DATA_BLOCK "DB_ProfinetDiagnostic"
TITLE = DB_ProfinetDiagnostic
{ S7_Optimized_Access := 'TRUE' }
AUTHOR : MHSE
FAMILY : GeneralSystemFunctions
VERSION : 3.0
NON_RETAIN
//Data block to store profinet network diagnostic data.
   VAR
      ProfinetNetworks { ExternalAccessible := 'False'; ExternalVisible := 'False'; ExternalWritable := 'False'; S7_SetPoint := 'False'} : Array[1..10] of "UDT_ProfinetNetwork";
   END_VAR


BEGIN

END_DATA_BLOCK

DATA_BLOCK "DI_OnOffDevices"
{ S7_Optimized_Access := 'TRUE' }
AUTHOR : MHSE
FAMILY : GeneralSystemFunctions
VERSION : 2.0
NON_RETAIN
"FB_OnOffDevices"

BEGIN

END_DATA_BLOCK

DATA_BLOCK "DB_Statistics"
TITLE = DB_Statistics
{ S7_Optimized_Access := 'TRUE' }
AUTHOR : MHSE
FAMILY : GeneralSystemFunctions
VERSION : 3.0
NON_RETAIN
//Data block to store statistical data.
   VAR
      Communication : Struct   // Communication statistic
         TCPIPConnect : "UDT_TCPIPConnectStatistics";   // TCPIP Connect statistics
         TCPIPReceive : "UDT_TCPIPReceiveStatistics";   // TCPIP Receive statistics
      END_STRUCT;
      System : Struct   // System statistic
         MCP { S7_SetPoint := 'False'} : "UDT_MainControlPanelStatistics";   // Statistics of Main Control Panel
         CPG01 : "UDT_ControlPowerGroupStatistics";   // Statistics of  Control Power Group 01
         CPG02 : "UDT_ControlPowerGroupStatistics";   // Statistics of  Control Power Group 02
         CPG03 : "UDT_ControlPowerGroupStatistics";   // Statistics of  Control Power Group 03
         CPG04 : "UDT_ControlPowerGroupStatistics";   // Statistics of  Control Power Group 04
         CPG05 : "UDT_ControlPowerGroupStatistics";   // Statistics of  Control Power Group 05
         Profinet { S7_SetPoint := 'False'} : "UDT_ProfiDiagStatistics";
      END_STRUCT;
   END_VAR


BEGIN

END_DATA_BLOCK

DATA_BLOCK "DB_FIFOMedPrioMsg"
TITLE = DB_FIFO
{ S7_Optimized_Access := 'TRUE' }
AUTHOR : MHSE
FAMILY : GeneralSystemFunctions
VERSION : 3.0
NON_RETAIN
//Data block to store FIFO registers.
   VAR RETAIN
      Header { ExternalAccessible := 'False'; ExternalVisible := 'False'; ExternalWritable := 'False'; S7_SetPoint := 'False'} : "UDT_FifoHeader";   // FIFO Header
      Data { ExternalAccessible := 'False'; ExternalVisible := 'False'; ExternalWritable := 'False'; S7_SetPoint := 'False'} : Array[0..199] of "UDT_Message";   // FIFO data buffer
   END_VAR


BEGIN

END_DATA_BLOCK

DATA_BLOCK "DB_FIFOLowPrioMsg"
TITLE = DB_FIFO
{ S7_Optimized_Access := 'TRUE' }
AUTHOR : MHSE
FAMILY : GeneralSystemFunctions
VERSION : 3.0
NON_RETAIN
//Data block to store FIFO registers.
   VAR RETAIN
      Header { ExternalAccessible := 'False'; ExternalVisible := 'False'; ExternalWritable := 'False'; S7_SetPoint := 'False'} : "UDT_FifoHeader";   // FIFO Header
      Data { ExternalAccessible := 'False'; ExternalVisible := 'False'; ExternalWritable := 'False'; S7_SetPoint := 'False'} : Array[0..199] of "UDT_Message";   // FIFO data buffer
   END_VAR


BEGIN

END_DATA_BLOCK

DATA_BLOCK "DB_FIFORcvMsg"
TITLE = DB_FIFO
{ S7_Optimized_Access := 'TRUE' }
AUTHOR : MHSE
FAMILY : GeneralSystemFunctions
VERSION : 3.0
NON_RETAIN
//Data block to store FIFO registers.
   VAR RETAIN
      Header { ExternalAccessible := 'False'; ExternalVisible := 'False'; ExternalWritable := 'False'; S7_SetPoint := 'False'} : "UDT_FifoHeader";   // FIFO Header
      Data { ExternalAccessible := 'False'; ExternalVisible := 'False'; ExternalWritable := 'False'; S7_SetPoint := 'False'} : Array[0..199] of "UDT_Message";   // FIFO data buffer
   END_VAR


BEGIN

END_DATA_BLOCK

DATA_BLOCK "DB_ParametrizationErrors"
TITLE = DB_ParametrizationErrors
{ S7_Optimized_Access := 'TRUE' }
AUTHOR : MHSE
FAMILY : GeneralSystemFunctions
VERSION : 3.0
NON_RETAIN
//Data block to store parametrization errors.
   VAR
      System { ExternalAccessible := 'False'; ExternalVisible := 'False'; ExternalWritable := 'False'} : Struct
         Communication { ExternalAccessible := 'False'; ExternalVisible := 'False'; ExternalWritable := 'False'} : Struct
            TCPIPSendError { ExternalAccessible := 'False'; ExternalVisible := 'False'; ExternalWritable := 'False'} : Bool;   // TCPIP send error
            TCPIPSendWarning { ExternalAccessible := 'False'; ExternalVisible := 'False'; ExternalWritable := 'False'} : Bool;   // TCPIP send warning
            TCPIPReceiveError { ExternalAccessible := 'False'; ExternalVisible := 'False'; ExternalWritable := 'False'} : Bool;   // TCPIP receive error
            TCPIPReceiveWarning { ExternalAccessible := 'False'; ExternalVisible := 'False'; ExternalWritable := 'False'} : Bool;   // TCPIP receive warning
         END_STRUCT;
      END_STRUCT;
   END_VAR


BEGIN

END_DATA_BLOCK

DATA_BLOCK "DB_CommonStatus"
TITLE = DB_Status
{ S7_Optimized_Access := 'TRUE' }
AUTHOR : MHSE
FAMILY : GeneralSystemFunctions
VERSION : 3.0
NON_RETAIN
//Data block to store status data.
   VAR
      Communication : Struct   // Communication status
         TCPIPConnect : "UDT_CommonStatus";   // FB_TCPIPConnect status
      END_STRUCT;
      System : Struct   // System statuses
         System1 { S7_SetPoint := 'False'} : "UDT_CommonStatus";
         MCP { S7_SetPoint := 'False'} : "UDT_CommonStatus";
         CPG01 : "UDT_CommonStatus";
         CPG02 : "UDT_CommonStatus";
         CPG03 : "UDT_CommonStatus";
         CPG04 : "UDT_CommonStatus";
         CPG05 : "UDT_CommonStatus";
         test { S7_SetPoint := 'True'} : Int;
      END_STRUCT;
   END_VAR


BEGIN

END_DATA_BLOCK

DATA_BLOCK "DB_Status"
TITLE = DB_Status
{ S7_Optimized_Access := 'TRUE' }
AUTHOR : MHSE
FAMILY : GeneralSystemFunctions
VERSION : 3.0
NON_RETAIN
//Data block to store status data.
   VAR
      Communication : Struct   // Communication status
         TCPIPConnect : "UDT_TCPIPConnectStatus";   // FB_TCPIPConnect status
      END_STRUCT;
      System : Struct   // System status
         MCP { S7_SetPoint := 'False'} : "UDT_MainControlPanelStatus";   // Status of Main Control Panel
         CPG01 : "UDT_ControlPowerGroupStatus";   // Status of  Control Power Group 01
         CPG02 : "UDT_ControlPowerGroupStatus";   // Status of  Control Power Group 02
         CPG03 : "UDT_ControlPowerGroupStatus";   // Status of  Control Power Group 03
         CPG04 : "UDT_ControlPowerGroupStatus";   // Status of  Control Power Group 04
         CPG05 : "UDT_ControlPowerGroupStatus";   // Status of  Control Power Group 05
         System1 : "UDT_SystemControlStatus";
      END_STRUCT;
   END_VAR


BEGIN

END_DATA_BLOCK

FUNCTION_BLOCK "FB_SoftVersion"
TITLE = FB_SoftVersion
{ S7_Optimized_Access := 'TRUE' }
AUTHOR : MHSE
FAMILY : GeneralSystemFunctions
VERSION : 3.0
// ATTRIBUTES
// AUTO_NUMBER = True
// BLOCK_NUMBER = 28
// END_ATTRIBUTES
//Function block to get the program checksums.
   VAR_INPUT
      is_ActualDateTime : String;   // Actual date and time
   END_VAR

   VAR_OUTPUT
      qs_SoftVersion : String[8];   // Software version
      qa_StandardCRC : Array[0..7] of Byte;   // Standard program checksum output
      qa_SafetyCRC : Array[0..7] of Byte;   // Safety program checksum output
   END_VAR

   VAR
      sFB_GetChecksum_Safety {InstructionName := 'GetChecksum'; LibVersion := '1.0'} : GetChecksum;   // Safety checksum read block
      sFB_GetChecksum_Standard {InstructionName := 'GetChecksum'; LibVersion := '1.0'} : GetChecksum;   // Standard checksum read block
   END_VAR
   VAR RETAIN
      sa_StandardCRC : Array[0..7] of Byte;   // Standard program checksum
      sa_SafetyCRC : Array[0..7] of Byte;   // Safety program checksum
   END_VAR
   VAR
      sa_NewStandardCRC { ExternalAccessible := 'False'; ExternalVisible := 'False'; ExternalWritable := 'False'} : Array[0..7] of Byte;   // New standard program checksum
      sa_NewSafetyCRC { ExternalAccessible := 'False'; ExternalVisible := 'False'; ExternalWritable := 'False'} : Array[0..7] of Byte;   // New safety program checksum
   END_VAR
   VAR RETAIN
      ss_Date { ExternalAccessible := 'False'; ExternalVisible := 'False'; ExternalWritable := 'False'} : String[8];   // Date charater string
   END_VAR

   VAR_TEMP
      ta_StandardCRC : Struct   // GetChecksum
         tx_Done : Bool;   // GetChecksum - Done
         tx_Busy : Bool;   // GetChecksum - Busy
         tx_Error : Bool;   // GetChecksum - Error
         tw_Status : Word;   // GetChecksum - Status
      END_STRUCT;
      ta_SafetyCRC : Struct   // GetChecksum
         tx_Done : Bool;   // GetChecksum - Done
         tx_Busy : Bool;   // GetChecksum - Busy
         tx_Error : Bool;   // GetChecksum - Error
         tw_Status : Word;   // GetChecksum - Status
      END_STRUCT;
      tx_CRCValid : Bool;   // Checksums valid
   END_VAR


BEGIN
	(*
	----------------------------------------------------------------------------------------

	Version history:
	Date        | Version   | Author        | Remark
	----------------------------------------------------------------------------------------
	24/05/2019  | 0.1       | K.Pokorski    | first release MHS TIA 15.1
	14/06/2019  | 0.2       | A.Nowak       | Replacement of instruction if for direct write into variable - Region 2
	24/07/2019  | 2.0       | L.Klar        | 2.0 MHS library release TIA 15.1
	27/08/2019  | 2.2       | K.Pokorski    | Comments adjusted
	12/11/2019  | 3.0       | P.Majka       | 3.0 MHS library release TIA 15.1
	21/02/2023  | 4.0       | F.Baten       | 4.0 Release TIA 17.5
	*)

	REGION 1 - Standard and safety program checksums

	    // Scope - 1 - Standard program CRC
	    #sFB_GetChecksum_Standard(Scope := 1,
	                              Done => #ta_StandardCRC.tx_Done,
	                              Busy => #ta_StandardCRC.tx_Busy,
	                              Error => #ta_StandardCRC.tx_Error,
	                              Status => #ta_StandardCRC.tw_Status,
	                              Checksum := #sa_NewStandardCRC);

	    // Scope - 2 - Safety program CRC
	    #sFB_GetChecksum_Safety(Scope := 2,
	                            Done => #ta_SafetyCRC.tx_Done,
	                            Busy => #ta_SafetyCRC.tx_Busy,
	                            Error => #ta_SafetyCRC.tx_Error,
	                            Status => #ta_SafetyCRC.tw_Status,
	                            Checksum := #sa_NewSafetyCRC);

	END_REGION

	REGION 2 - Checksums comparison

	    #tx_CRCValid := (#sa_NewStandardCRC = #sa_StandardCRC)
	    AND (#sa_SafetyCRC = #sa_NewSafetyCRC);

	END_REGION

	REGION 3 - New software version

	    // Separate the year, mounth and day from actual date and time and connect it to one string
	    IF (NOT #tx_CRCValid)                                           // Checksums not valid
	    THEN

	        #ss_Date := CONCAT(IN1 := MID(IN := #is_ActualDateTime,
	                                                         L := 4,
	                                                         P := 1),

	                           IN2 := MID(IN := #is_ActualDateTime,
	                                      L := 2,
	                                      P := 6),

	                           IN3 := MID(IN := #is_ActualDateTime,
	                                      L := 2,
	                                      P := 9));

	        // Standard progrm checksum update
	        #sa_StandardCRC := #sa_NewStandardCRC;

	        // Safety program checksum update
	        #sa_SafetyCRC := #sa_NewSafetyCRC;

	    END_IF;

	END_REGION

	REGION 4 - Write outputs

	    // New program date
	    #qs_SoftVersion := #ss_Date;

	    // Actual standard program checksum
	    #qa_StandardCRC := #sa_StandardCRC;

	    // Actual safety program checksum
	    #qa_SafetyCRC := #sa_SafetyCRC;

	END_REGION
END_FUNCTION_BLOCK

DATA_BLOCK "DB_Configuration"
TITLE = DB_Configuration
{ S7_Optimized_Access := 'TRUE' }
AUTHOR : MHSE
FAMILY : GeneralSystemFunctions
VERSION : 3.0
NON_RETAIN
//Data block to store configuration data.
   VAR RETAIN
      System { ExternalAccessible := 'False'; ExternalVisible := 'False'; ExternalWritable := 'False'} : Struct   // System configuration
         Connection { ExternalAccessible := 'False'; ExternalVisible := 'False'; ExternalWritable := 'False'} : "UDT_Connection";   // Connection configuration
      END_STRUCT;
   END_VAR


BEGIN
   System.Connection.ActiveEstablished := TRUE;
   System.Connection.Interface_ID := 64;
   System.Connection.ID := 16#0001;
   System.Connection.IP[1] := 192;
   System.Connection.IP[2] := 168;
   System.Connection.IP[3] := 3;
   System.Connection.IP[4] := 53;
   System.Connection.Port := 42300;
   System.Connection.ConTimeout := 5000;

END_DATA_BLOCK

FUNCTION_BLOCK "FB_ProfiDiag"
TITLE = FB_ProfiDiag
{ S7_Optimized_Access := 'TRUE' }
AUTHOR : MHSE
FAMILY : GeneralSystemFunctions
VERSION : 3.0
// ATTRIBUTES
// AUTO_NUMBER = True
// BLOCK_NUMBER = 25
// END_ATTRIBUTES
//Function block to diagnose Profinet network.
   VAR_INPUT
      iui_LADDR : HW_IOSYSTEM;   // Hardware identifier of the PROFINET IO
      ix_ExternalScan { ExternalAccessible := 'False'; ExternalVisible := 'False'; ExternalWritable := 'False'} : Bool;   // External scan
   END_VAR

   VAR_OUTPUT
      qx_ProfinetOk { ExternalAccessible := 'False'; ExternalVisible := 'False'; ExternalWritable := 'False'} : Bool;   // Profinet ok
      qx_Error { ExternalAccessible := 'False'; ExternalVisible := 'False'; ExternalWritable := 'False'} : Bool;   // Collective error output
   END_VAR

   VAR_IN_OUT
      iqUDT_EquipmentControl : "UDT_EquipmentControl";   // Equipment control structure
      iqUDT_PNDiagArray : "UDT_ProfinetNetwork";   // Profinet devices status array
      iqUDT_Statistics : "UDT_ProfiDiagStatistics";   // Statistics structure
   END_VAR

   VAR
      s_GetProjectName {InstructionName := 'Get_Name'; LibVersion := '1.3'} : Get_Name;   // Get name function
      sa_Status : Struct   // Status structure
         ErrorCode : Struct   // Error code structure
            DeviceState : Int;   // Siemens "DeviceState" error code
            GEO2LOG : Int;   // Siemens "GEO2LOG" error code
            LOG2GEO : Int;   // Siemens "LOG2GEO" error code
            GetName : Word;   // Siemens "GetName" error code
         END_STRUCT;
      END_STRUCT;
      sx_PNOK : Bool := FALSE;   // Profinet OK
      sx_NewEvent { ExternalAccessible := 'False'; ExternalVisible := 'False'; ExternalWritable := 'False'} : Bool;   // New event
   END_VAR

   VAR_TEMP
      tv_ProfinetGeoAdr {InstructionName := 'GEOADDR'; LibVersion := '1.0'} : GEOADDR;   // Profinet network geo structure
      tv_DeviceGeoAdr {InstructionName := 'GEOADDR'; LibVersion := '1.0'} : GEOADDR;   // Profinet device geo structure
      ta_Configured : Array[0..1024] of Bool;   // Configured devices array
      ta_Exist : Array[0..1024] of Bool;   // Existing devices array
      ta_Error : Array[0..1024] of Bool;   // Devices errors array
      ti_DeviceNr : Int;   // Device number
      ti_NrOfDevicesError : Int;   // Number of devices error
      ti_DiagArraySize : Int;   // Diagnostic array size
   END_VAR

   VAR CONSTANT
      cui_ConfiguredDevicesMode : UInt := 1;   // Scan mode of configured devices
      cui_ExistingDevicesMode : UInt := 4;   // Scan mode of existing devices
      cui_DevicesErrorMode : UInt := 2;   // Scan mode of devices error
      cui_HWType : UInt := 2;   // IO device hardware type
      cui_Area : UInt := 1;   // IO device area
   END_VAR


BEGIN
	(*
	----------------------------------------------------------------------------------------

	Version history:
	Date        | Version   | Author        | Remark
	----------------------------------------------------------------------------------------
	24/05/2019  | 0.1       | K.Pokorski    | first release MHS TIA 15.1
	13/06/2019  | 0.2       | A.Nowak       | Replacement of instruction if for direct write into variable - Region 3
	24/06/2019  | 0.3       | L.Klar        | Status running added
	19/07/2019  | 0.5       | L.Klar        | Status handling changed, output qx_ProfinetOk added
	24/07/2019  | 2.0       | L.Klar        | 2.0 MHS library release TIA 15.1
	14/08/2019  | 2.1       | K.Pokorski    | HW_ID and TIA device project name handling added
	26/08/2019  | 2.2       | K.Pokorski    | Comments adjusted
	20/09/2019  | 2.3       | K.Pokorski    | "UDT_Status" deleted
	04/11/2019  | 2.4       | L.Klar        | Scan profinet and first scan changed from memory bit to DB variable
	12/11/2019  | 3.0       | P.Majka       | 3.0 MHS library release TIA 15.1
	21/02/2023  | 4.0       | F.Baten       | 4.0 Release TIA 17.5
	*)

	REGION 1 – Scan request

	    IF ("DB_Memory".ScanProfinet    // Scan request from diagnostic OB
	        OR "DB_Memory".FirstScan    // First PLC cycle
	        OR #ix_ExternalScan)        // External scan available
	    THEN

	        #sx_PNOK := FALSE;

	    END_IF;

	END_REGION

	REGION 2 – Devices states update

	    // Scan devices, extract device status: configured, exists, error when profinet network not ok
	    IF (NOT #sx_PNOK)       // Profinet needs a scan
	    THEN

	        #sa_Status.ErrorCode.DeviceState := DeviceStates(LADDR := #iui_LADDR,
	                                                         MODE := #cui_ConfiguredDevicesMode,
	                                                         STATE := #ta_Configured);

	        #sa_Status.ErrorCode.DeviceState := DeviceStates(LADDR := #iui_LADDR,
	                                                         MODE := #cui_ExistingDevicesMode,
	                                                         STATE := #ta_Exist);

	        #sa_Status.ErrorCode.DeviceState := DeviceStates(LADDR := #iui_LADDR,
	                                                         MODE := #cui_DevicesErrorMode,
	                                                         STATE := #ta_Error);

	    END_IF;

	END_REGION

	REGION 3 – Devices Statuses update

	    // Move device state to diagnostic structure if network required scan and no error occured during scan
	    IF (NOT #sx_PNOK                                                                                                    // Profinet not ok
	        AND #sa_Status.ErrorCode.DeviceState = 0)                                                                       // "DeviceStates" error free
	    THEN

	        // Initialise reset device errors counter
	        #ti_NrOfDevicesError := 0;

	        // Maximum number of Profinet devices
	        #ti_DiagArraySize := "FC_GetNrOfArrayEl"(iv_Array := #iqUDT_PNDiagArray.DeviceStatus);

	        // A loop operating on Profinet devices
	        FOR #ti_DeviceNr := 0 TO (#ti_DiagArraySize - 1)
	        DO

	            // The device is configured in TIA Portal
	            IF (#ta_Configured[#ti_DeviceNr])                                                                           // Devices configured
	            THEN

	                // Set the device configured status bit in diagnostic structure
	                #iqUDT_PNDiagArray.DeviceStatus[#ti_DeviceNr].DeviceState.Configure := TRUE;

	                // Move device profinet number to diagnostic structure
	                #iqUDT_PNDiagArray.DeviceStatus[#ti_DeviceNr].DeviceState.ProfinetNumber := INT_TO_UINT(#ti_DeviceNr);

	                // Get the Profinet network IOSystem address
	                #sa_Status.ErrorCode.LOG2GEO := LOG2GEO(LADDR := #iui_LADDR, GEOADDR := #tv_ProfinetGeoAdr);

	                // Configuring parameters for extracting the device's HW_ID
	                #tv_DeviceGeoAdr.HWTYPE := #cui_HWType;
	                #tv_DeviceGeoAdr.AREA := #cui_Area;
	                #tv_DeviceGeoAdr.STATION := INT_TO_UINT(#ti_DeviceNr);
	                #tv_DeviceGeoAdr.IOSYSTEM := #tv_ProfinetGeoAdr.IOSYSTEM;

	                // Extracting the device's HW_ID
	                #sa_Status.ErrorCode.GEO2LOG := GEO2LOG(GEOADDR := #tv_DeviceGeoAdr,
	                                                        LADDR => #iqUDT_PNDiagArray.DeviceStatus[#ti_DeviceNr].DeviceState.HW_ID);

	                // Move device's project name to diagnostic structure
	                #s_GetProjectName(LADDR := #iui_LADDR,
	                                  STATION_NR := INT_TO_UINT(#ti_DeviceNr),
	                                  STATUS => #sa_Status.ErrorCode.GetName,
	                                  DATA := #iqUDT_PNDiagArray.DeviceStatus[#ti_DeviceNr].DeviceState.PNDeviceName);

	                // Move device exist state to the Profinet diagnostic structure
	                IF (#ta_Exist[#ti_DeviceNr])                                                                                // Device exist
	                THEN

	                    #iqUDT_PNDiagArray.DeviceStatus[#ti_DeviceNr].DeviceState.Exist := TRUE;

	                ELSE

	                    #iqUDT_PNDiagArray.DeviceStatus[#ti_DeviceNr].DeviceState.Exist := FALSE;

	                    // Increment the number of devices error
	                    #ti_NrOfDevicesError += 1;

	                END_IF;
	                // Move device error state to the Profinet diagnostic structure
	                IF (NOT #ta_Error[#ti_DeviceNr])                                                                            // Device is error free
	                THEN

	                    #iqUDT_PNDiagArray.DeviceStatus[#ti_DeviceNr].DeviceState.Error := FALSE;

	                ELSE

	                    // New error detected
	                    #sx_NewEvent := NOT #iqUDT_PNDiagArray.DeviceStatus[#ti_DeviceNr].DeviceState.Error;

	                    // Statistics handling
	                    IF (#ta_Error[#ti_DeviceNr]                                                                             // Device has error
	                        OR #iqUDT_EquipmentControl.Command.ResetData)                                                      // Reset statistics available
	                    THEN

	                        "FC_Statistics"(ix_Reset := #iqUDT_EquipmentControl.Command.ResetData,
	                                        ix_Activate := #ta_Error[#ti_DeviceNr],
	                                        ix_RTrigActivate := #sx_NewEvent,
	                                        iqUDT_Statistics := #iqUDT_Statistics.DeviceError[#ti_DeviceNr]);

	                    END_IF;

	                    #iqUDT_PNDiagArray.DeviceStatus[#ti_DeviceNr].DeviceState.Error := TRUE;

	                    // Increment number of devices error
	                    #ti_NrOfDevicesError += 1;

	                END_IF;

	                // Reset all diagnostic information if the device is not configured in TIA Portal
	            ELSE

	                #iqUDT_PNDiagArray.DeviceStatus[#ti_DeviceNr].DeviceState.Configure := FALSE;
	                #iqUDT_PNDiagArray.DeviceStatus[#ti_DeviceNr].DeviceState.Exist := FALSE;
	                #iqUDT_PNDiagArray.DeviceStatus[#ti_DeviceNr].DeviceState.Error := FALSE;
	                #iqUDT_PNDiagArray.DeviceStatus[#ti_DeviceNr].DeviceState.HW_ID := 0;
	                #iqUDT_PNDiagArray.DeviceStatus[#ti_DeviceNr].DeviceState.ProfinetNumber := 0;
	                #iqUDT_PNDiagArray.DeviceStatus[#ti_DeviceNr].DeviceState.PNDeviceName := '';

	            END_IF;

	        END_FOR;

	    END_IF;

	END_REGION

	REGION 4 – Profinet OK

	    // Reset profinet error
	    IF (#ti_NrOfDevicesError = 0                        // Number of devices error equal to zero
	        AND (#iqUDT_EquipmentControl.Command.Reset     // Error reset required
	        OR #ix_ExternalScan))                           // External scan active
	    THEN

	        #sx_PNOK := TRUE;

	    END_IF;

	END_REGION

	REGION 5 – Status

	    // Update Profinet ok output status
	    #qx_ProfinetOk := #sx_PNOK;

	    // Create the collective block error bit
	    #qx_Error := #sa_Status.ErrorCode.DeviceState <> 0       // Profinet network error
	    OR #sa_Status.ErrorCode.GEO2LOG <> 0                     // "Geo2Log" standard Siemens block error
	    OR #sa_Status.ErrorCode.LOG2GEO <> 0                     // "Log2Geo" standard Siemens block error
	    OR #sa_Status.ErrorCode.GetName > 16#8000;               // "GetName" standard Siemens block error

	END_REGION
END_FUNCTION_BLOCK

FUNCTION "FC_Simulation" : Void
TITLE = FC_Simulation
{ S7_Optimized_Access := 'TRUE' }
AUTHOR : MHSE
FAMILY : GeneralSystemFunctions
VERSION : 3.0
// ATTRIBUTES
// AUTO_NUMBER = True
// BLOCK_NUMBER = 13
// END_ATTRIBUTES
//Function to enable simulation mode.
   VAR_TEMP
      tx_Done : Bool;
      tx_Error : Bool;
   END_VAR


BEGIN
	(*
	----------------------------------------------------------------------------------------

	Version history:
	Date        | Version   | Author        | Remark
	----------------------------------------------------------------------------------------
	24/05/2019  | 0.1       | L.Klar        | first release MHS TIA 15.1
	24/07/2019  | 2.0       | L.Klar        | 2.0 MHS library release TIA 15.1
	04/11/2019  | 2.1       | L.Klar        | Simulation bit changed from memory to DB variable
	12/11/2019  | 3.0       | P.Majka       | 3.0 MHS library release TIA 15.1
	21/02/2023  | 4.0       | F.Baten       | 4.0 Release TIA 17.5
	*)

	REGION 1 - Disabling and Enabling devices

	    "DI_OnOffDevices"(ix_Simulation := "DB_Memory".Simulation,
	                      qx_Done => #tx_Done,
	                      qx_Error => #tx_Error,
	                      iqa_ProfinetNetworks := "DB_ProfinetDiagnostic".ProfinetNetworks);

	END_REGION



END_FUNCTION

FUNCTION "FC_TimeToString" : Void
TITLE = FC_TimeToString
{ S7_Optimized_Access := 'TRUE' }
AUTHOR : MHSE
FAMILY : GeneralSystemFunctions
VERSION : 3.0
// ATTRIBUTES
// AUTO_NUMBER = True
// BLOCK_NUMBER = 29
// END_ATTRIBUTES
//Function to convert date in DTL to the string format.
   VAR_INPUT
      ia_Date {InstructionName := 'DTL'; LibVersion := '1.0'} : DTL;   // DTL format date
   END_VAR

   VAR_OUTPUT
      qs_Date : String;   // String format date
   END_VAR

   VAR_TEMP
      ta_StringDate : Struct   // String format date
         Year : String;   //   Year
         Month : String[2];   //   Month
         Day : String[2];   //   Day
         Hour : String[2];   //   Hour
         Minute : String[2];   //   Minunte
         Second : String[2];   //   Second
         Millisecond : String[4];   //   Millisecond
      END_STRUCT;
      ta_HTAReturn : Struct   // HTA operation status
         Year : Word;   //   Year
         Month : Word;   //   Month
         Day : Word;   //   Day
         Hour : Word;   //   Hour
         Minute : Word;   //   Minunte
         Second : Word;   //   Second
         Millisecond : Word;   //   Millisecond
      END_STRUCT;
   END_VAR

   VAR CONSTANT
      ci_Positions4 : USInt := 4;   // Number of character positions
      ci_DecimalPlaces0 : USInt := 0;   // Number of decimal places
      ci_Format0 : USInt := 0;   // Output format of the characters
      ci_Position1 : USInt := 1;   // Character starting at which the result is written
      cc_Colon : Char := ':';   // Colon sign
   END_VAR


BEGIN
	(*
	----------------------------------------------------------------------------------------

	Version history:
	Date        | Version   | Author        | Remark
	----------------------------------------------------------------------------------------
	24/05/2019  | 0.1       | K.Pokorski    | first release MHS TIA 15.1
	24/07/2019  | 2.0       | L.Klar        | 2.0 MHS library release TIA 15.1
	27/08/2019  | 2.1       | M.Kurpiers    | Comments adjusted
	05/09/2019  | 2.2       | K.Pokorski    | FC changed from unoptimized to optimized
	12/11/2019  | 3.0       | P.Majka       | 3.0 MHS library release TIA 15.1
	16/02/2023  | 3.1       | F.Baten       | Added constants
	21/02/2023  | 4.0       | F.Baten       | 4.0 Release TIA 17.5
	*)

	REGION 1 - Date and time separation

	    // Convert the year into a character string
	    VAL_STRG(IN := #ia_Date.YEAR,
	             SIZE := #ci_Positions4,
	             PREC := #ci_DecimalPlaces0,
	             FORMAT := USINT_TO_WORD(#ci_Format0),
	             P := #ci_Position1,
	             OUT => #ta_StringDate.Year);

	    // Using the HTA function, convert date into a string format
	    #ta_HTAReturn.Month := HTA(IN := WORD_TO_BYTE(INT_TO_BCD16((USINT_TO_INT(#ia_Date.MONTH)))), N := 1, OUT => #ta_StringDate.Month);                          // Convert the month
	    #ta_HTAReturn.Day := HTA(IN := WORD_TO_BYTE(INT_TO_BCD16((USINT_TO_INT(#ia_Date.DAY)))), N := 1, OUT => #ta_StringDate.Day);                                // Convert the day
	    #ta_HTAReturn.Hour := HTA(IN := WORD_TO_BYTE(INT_TO_BCD16((USINT_TO_INT(#ia_Date.HOUR)))), N := 1, OUT => #ta_StringDate.Hour);                             // Convert the hour
	    #ta_HTAReturn.Minute := HTA(IN := WORD_TO_BYTE(INT_TO_BCD16((USINT_TO_INT(#ia_Date.MINUTE)))), N := 1, OUT => #ta_StringDate.Minute);                       // Convert the minute
	    #ta_HTAReturn.Second := HTA(IN := WORD_TO_BYTE(INT_TO_BCD16((USINT_TO_INT(#ia_Date.SECOND)))), N := 1, OUT => #ta_StringDate.Second);                       // Convert the second
	    #ta_HTAReturn.Millisecond := HTA(IN := INT_TO_BCD16((UDINT_TO_INT(#ia_Date.NANOSECOND / 1000000))), N := 2, OUT => #ta_StringDate.Millisecond);              // Convert the millisecond

	END_REGION

	REGION 2 - Timestamp preparation

	    // Combine several input strings into one long output string
	    #qs_Date := (CONCAT(IN1 := #ta_StringDate.Year,
	                        IN2 := #cc_Colon,
	                        IN3 := #ta_StringDate.Month,
	                        IN4 := #cc_Colon,
	                        IN5 := #ta_StringDate.Day,
	                        IN6 := #cc_Colon,
	                        IN7 := #ta_StringDate.Hour,
	                        IN8 := #cc_Colon,
	                        IN9 := #ta_StringDate.Minute,
	                        IN10 := #cc_Colon,
	                        IN11 := #ta_StringDate.Second,
	                        IN12 := #cc_Colon,
	                        IN13 := RIGHT(IN := #ta_StringDate.Millisecond, L := 3)));

	END_REGION
END_FUNCTION

DATA_BLOCK "DI_TCPIPReceive"
{ S7_Optimized_Access := 'TRUE' }
VERSION : 0.1
NON_RETAIN
"FB_TCPIPReceive"

BEGIN

END_DATA_BLOCK

DATA_BLOCK "DB_Time"
TITLE = DB_Time
{ S7_Optimized_Access := 'TRUE' }
AUTHOR : MHSE
FAMILY : GeneralSystemFunctions
VERSION : 3.0
NON_RETAIN
//Data block to store date and time data.
   VAR
      ActualTimeDTL {InstructionName := 'DTL'; LibVersion := '1.0'; ExternalAccessible := 'False'; ExternalVisible := 'False'; ExternalWritable := 'False'} : DTL;   // Actual date and time in DTL
      ActualTime { ExternalAccessible := 'False'; ExternalVisible := 'False'; ExternalWritable := 'False'} : String;   // Actual date and time in String
      Timestamp { ExternalAccessible := 'False'; ExternalVisible := 'False'; ExternalWritable := 'False'} : String[17];   // Actual date and time in String
      DaylightSaving { ExternalAccessible := 'False'; ExternalVisible := 'False'; ExternalWritable := 'False'} : Int;
   END_VAR


BEGIN

END_DATA_BLOCK

DATA_BLOCK "DI_TCPIPSend"
{ S7_Optimized_Access := 'TRUE' }
VERSION : 0.1
NON_RETAIN
"FB_TCPIPSend"

BEGIN

END_DATA_BLOCK

DATA_BLOCK "DB_SoftwareVersion"
TITLE = DB_SoftwareVersion
{ S7_Optimized_Access := 'TRUE' }
AUTHOR : MHSE
FAMILY : GeneralSystemFunctions
VERSION : 3.0
NON_RETAIN
//Data block to store software version data.
   VAR
      "Version" { ExternalAccessible := 'False'; ExternalVisible := 'False'; ExternalWritable := 'False'} : String[8];   // Software version
      StandardChecksum { ExternalAccessible := 'False'; ExternalVisible := 'False'; ExternalWritable := 'False'} : Array[0..7] of Byte;   // Standard program checksum
      SafetyChecksum { ExternalAccessible := 'False'; ExternalVisible := 'False'; ExternalWritable := 'False'} : Array[0..7] of Byte;   // Safety program checksum
   END_VAR


BEGIN

END_DATA_BLOCK

DATA_BLOCK "DB_Control"
{ S7_Optimized_Access := 'TRUE' }
AUTHOR : MHSE
FAMILY : Equimpent
VERSION : 0.1
NON_RETAIN
   VAR
      System1 { ExternalAccessible := 'False'; ExternalVisible := 'False'; ExternalWritable := 'False'; S7_SetPoint := 'False'} : "UDT_EquipmentControl";
   END_VAR


BEGIN

END_DATA_BLOCK

DATA_BLOCK "DB_FIFOHighPrioMsg"
TITLE = DB_FIFO
{ S7_Optimized_Access := 'TRUE' }
AUTHOR : MHSE
FAMILY : GeneralSystemFunctions
VERSION : 3.0
NON_RETAIN
//Data block to store FIFO registers.
   VAR
      Header { ExternalAccessible := 'False'; ExternalVisible := 'False'; ExternalWritable := 'False'; S7_SetPoint := 'False'} : "UDT_FifoHeader";   // FIFO Header
      Data { ExternalAccessible := 'False'; ExternalVisible := 'False'; ExternalWritable := 'False'; S7_SetPoint := 'False'} : Array[0..199] of "UDT_Message";   // FIFO data buffer
   END_VAR


BEGIN

END_DATA_BLOCK

DATA_BLOCK "DI_TCPIPConnect"
{ S7_Optimized_Access := 'TRUE' }
VERSION : 0.1
NON_RETAIN
"FB_TCPIPConnect"

BEGIN

END_DATA_BLOCK

FUNCTION_BLOCK "FB_SystemFunctions"
TITLE = FB_SystemFunctions
{ S7_Optimized_Access := 'TRUE' }
AUTHOR : MHSE
FAMILY : GeneralSystemFunctions
VERSION : 3.0
// ATTRIBUTES
// AUTO_NUMBER = True
// BLOCK_NUMBER = 200
// END_ATTRIBUTES
//Function to execute system functions.
   VAR
      sFB_SoftVersion { ExternalAccessible := 'False'; ExternalVisible := 'False'; ExternalWritable := 'False'; S7_SetPoint := 'False'} : "FB_SoftVersion";   // Software version block instance
      sFB_ProfiDiag_Net1 { ExternalAccessible := 'False'; ExternalVisible := 'False'; ExternalWritable := 'False'; S7_SetPoint := 'False'} : "FB_ProfiDiag";   // Profinet diagnostic block instance
      sFB_ProfiDiag_Net2 { ExternalAccessible := 'False'; ExternalVisible := 'False'; ExternalWritable := 'False'; S7_SetPoint := 'False'} : "FB_ProfiDiag";   // Profinet diagnostic block instance
      sFB_ProfiDiag_Net3 { ExternalAccessible := 'False'; ExternalVisible := 'False'; ExternalWritable := 'False'; S7_SetPoint := 'False'} : "FB_ProfiDiag";   // Profinet diagnostic block instance
      sFB_ProfiDiag_Net4 { ExternalAccessible := 'False'; ExternalVisible := 'False'; ExternalWritable := 'False'; S7_SetPoint := 'False'} : "FB_ProfiDiag";   // Profinet diagnostic block instance
      sFB_ProfiDiag_Net5 { ExternalAccessible := 'False'; ExternalVisible := 'False'; ExternalWritable := 'False'; S7_SetPoint := 'False'} : "FB_ProfiDiag";   // Profinet diagnostic block instance
      sFB_ProfiDiag_Net6 { ExternalAccessible := 'False'; ExternalVisible := 'False'; ExternalWritable := 'False'; S7_SetPoint := 'False'} : "FB_ProfiDiag";   // Profinet diagnostic block instance
      sFB_ProfiDiag_Net7 { ExternalAccessible := 'False'; ExternalVisible := 'False'; ExternalWritable := 'False'; S7_SetPoint := 'False'} : "FB_ProfiDiag";   // Profinet diagnostic block instance
      sFB_ProfiDiag_Net8 { ExternalAccessible := 'False'; ExternalVisible := 'False'; ExternalWritable := 'False'; S7_SetPoint := 'False'} : "FB_ProfiDiag";   // Profinet diagnostic block instance
      sFB_ProfiDiag_Net9 { ExternalAccessible := 'False'; ExternalVisible := 'False'; ExternalWritable := 'False'; S7_SetPoint := 'False'} : "FB_ProfiDiag";   // Profinet diagnostic block instance
      sFB_ProfiDiag_Net10 { ExternalAccessible := 'False'; ExternalVisible := 'False'; ExternalWritable := 'False'; S7_SetPoint := 'False'} : "FB_ProfiDiag";   // Profinet diagnostic block instance
      sR_TRIG0_1Sec {InstructionName := 'R_TRIG'; LibVersion := '1.0'; ExternalAccessible := 'False'; ExternalVisible := 'False'; ExternalWritable := 'False'; S7_SetPoint := 'False'} : R_TRIG;   // Rise trigger to detect edge each 0.1 second
      sR_TRIG0_2Sec {InstructionName := 'R_TRIG'; LibVersion := '1.0'; ExternalAccessible := 'False'; ExternalVisible := 'False'; ExternalWritable := 'False'; S7_SetPoint := 'False'} : R_TRIG;   // Rise trigger to detect edge each 0.2 second
      sR_TRIG0_4Sec {InstructionName := 'R_TRIG'; LibVersion := '1.0'; ExternalAccessible := 'False'; ExternalVisible := 'False'; ExternalWritable := 'False'; S7_SetPoint := 'False'} : R_TRIG;   // Rise trigger to detect edge each 0.4 second
      sR_TRIG0_5Sec {InstructionName := 'R_TRIG'; LibVersion := '1.0'; ExternalAccessible := 'False'; ExternalVisible := 'False'; ExternalWritable := 'False'; S7_SetPoint := 'False'} : R_TRIG;   // Rise trigger to detect edge each 0.5 second
      sR_TRIG0_8Sec {InstructionName := 'R_TRIG'; LibVersion := '1.0'; ExternalAccessible := 'False'; ExternalVisible := 'False'; ExternalWritable := 'False'; S7_SetPoint := 'False'} : R_TRIG;   // Rise trigger to detect edge each 0.8 second
      sR_TRIG_1Sec {InstructionName := 'R_TRIG'; LibVersion := '1.0'; ExternalAccessible := 'False'; ExternalVisible := 'False'; ExternalWritable := 'False'; S7_SetPoint := 'False'} : R_TRIG;   // Rise trigger to detect edge each 1 second
      sR_TRIG1_6Sec {InstructionName := 'R_TRIG'; LibVersion := '1.0'; ExternalAccessible := 'False'; ExternalVisible := 'False'; ExternalWritable := 'False'; S7_SetPoint := 'False'} : R_TRIG;   // Rise trigger to detect edge each 1.6 second
      sR_TRIG_2Sec {InstructionName := 'R_TRIG'; LibVersion := '1.0'; ExternalAccessible := 'False'; ExternalVisible := 'False'; ExternalWritable := 'False'; S7_SetPoint := 'False'} : R_TRIG;   // Rise trigger to detect edge each 2 second
   END_VAR
   VAR DB_SPECIFIC
      sx_Reset { ExternalAccessible := 'False'; ExternalVisible := 'False'; ExternalWritable := 'False'} : Bool;   // Profinet fault reset
      sx_ResetData { ExternalAccessible := 'False'; ExternalVisible := 'False'; ExternalWritable := 'False'} : Bool;   // Profinet statistic data reset
   END_VAR
   VAR
      sx_Error { ExternalAccessible := 'False'; ExternalVisible := 'False'; ExternalWritable := 'False'} : Bool;
      sx_ProfiDiag_Net1_OK { ExternalAccessible := 'False'; ExternalVisible := 'False'; ExternalWritable := 'False'} : Bool;   // Profinet network 1 Ok
      sx_ProfiDiag_Net2_OK { ExternalAccessible := 'False'; ExternalVisible := 'False'; ExternalWritable := 'False'} : Bool;   // Profinet network 2 Ok
      sx_ProfiDiag_Net3_OK { ExternalAccessible := 'False'; ExternalVisible := 'False'; ExternalWritable := 'False'} : Bool;   // Profinet network 3 Ok
      sx_ProfiDiag_Net4_OK { ExternalAccessible := 'False'; ExternalVisible := 'False'; ExternalWritable := 'False'} : Bool;   // Profinet network 4 Ok
      sx_ProfiDiag_Net5_OK { ExternalAccessible := 'False'; ExternalVisible := 'False'; ExternalWritable := 'False'} : Bool;   // Profinet network 5 Ok
      sx_ProfiDiag_Net6_OK { ExternalAccessible := 'False'; ExternalVisible := 'False'; ExternalWritable := 'False'} : Bool;   // Profinet network 6 Ok
      sx_ProfiDiag_Net7_OK { ExternalAccessible := 'False'; ExternalVisible := 'False'; ExternalWritable := 'False'} : Bool;   // Profinet network 7 Ok
      sx_ProfiDiag_Net8_OK { ExternalAccessible := 'False'; ExternalVisible := 'False'; ExternalWritable := 'False'} : Bool;   // Profinet network 8 Ok
      sx_ProfiDiag_Net9_OK { ExternalAccessible := 'False'; ExternalVisible := 'False'; ExternalWritable := 'False'} : Bool;   // Profinet network 9 Ok
      sx_ProfiDiag_Net10_OK { ExternalAccessible := 'False'; ExternalVisible := 'False'; ExternalWritable := 'False'} : Bool;   // Profinet network 10 Ok
   END_VAR

   VAR_TEMP
      tui_LADDR : HW_IOSYSTEM;
      tUDT_EquipmentControl : "UDT_EquipmentControl";
      ti_RD_LOC_T_Status : Int;   // RD_LOC_T - Read actual date and time function status
      tx_replace : Bool;
   END_VAR


BEGIN
	(*
	----------------------------------------------------------------------------------------
	|                                                                                      |
	|  Copyright  2019             MHS                                                     |
	|  All Rights Reserved         Larenweg 90                                             |
	|                              5234 KC 's-Hertogenbosch,                               |
	|                              Netherlands                                             |
	|                                                                                      |
	----------------------------------------------------------------------------------------

	Version history:
	Date        | Version   | Author        | Remark
	----------------------------------------------------------------------------------------
	24/05/2019  | 0.1       | L.Klar        | first release MHS TIA 15.1
	24/07/2019  | 2.0       | L.Klar        | 2.0 MHS library release TIA 15.1
	03/10/2019  | 2.1       | L.Klar        | Comments adjusted
	04/10/2019  | 2.2       | L.Klar        | profinet scan marker reset added
	30/10/2019  | 2.3       | S.Theocharis  | Update the PN calls
	04/11/2019  | 2.4       | L.Klar        | Memory bits changed to DB variables
	12/11/2019  | 3.0       | P.Majka       | 3.0 MHS library release TIA 15.1
	11/12/2019  | 3.1       | S. Deulkar    | Called FC simulation in region 2
	21/02/2023  | 4.0       | F.Baten       | 4.0 Release TIA 17.5
	*)

	REGION 1 – PLC scan cycle measurement

	    "DB_Memory".PrevCycleTime := RUNTIME("DB_Memory".RuntimeMem) * 1000;

	END_REGION

	REGION 2 – Simulation

	    "FC_Simulation"();

	END_REGION

	REGION 3 – One shot of PLC clock pulse

	    // One shot every 0.1 sec of 10 Hz clock memory
	    #sR_TRIG0_1Sec(CLK := "DB_Memory".Clock_10Hz,
	                   Q => "DB_Memory"."OS_0.1sec");

	    // One shot every 0.2 sec of 5 Hz clock memory
	    #sR_TRIG0_2Sec(CLK := "DB_Memory".Clock_5Hz,
	                   Q => "DB_Memory"."OS_0.2sec");

	    // One shot every 0.4 sec of 2.5 Hz clock memory
	    #sR_TRIG0_4Sec(CLK := "DB_Memory"."Clock_2.5Hz",
	                   Q => "DB_Memory"."OS_0.4sec");

	    // One shot every 0.5 sec of 2 Hz clock memory
	    #sR_TRIG0_5Sec(CLK := "DB_Memory".Clock_2Hz,
	                   Q => "DB_Memory"."OS_0.5sec");

	    // One shot every 0.8 sec of 1.25 Hz clock memory
	    #sR_TRIG0_8Sec(CLK := "DB_Memory"."Clock_1.25Hz",
	                   Q => "DB_Memory"."OS_0.8sec");

	    // One shot every 1 sec of 1 Hz clock memory
	    #sR_TRIG_1Sec(CLK := "DB_Memory".Clock_1Hz,
	                  Q => "DB_Memory".OS_1sec);

	    // One shot every 1.6 sec of 0.625 Hz clock memory
	    #sR_TRIG1_6Sec(CLK := "DB_Memory"."Clock_0.625Hz",
	                   Q => "DB_Memory"."OS_1.6sec");

	    // One shot every 2 sec of 0.5 Hz clock memory
	    #sR_TRIG_2Sec(CLK := "DB_Memory"."Clock_0.5Hz",
	                  Q => "DB_Memory".OS_2sec);


	END_REGION

	REGION 4 – Actual time

	    // Read actual PLC date and time
	    #ti_RD_LOC_T_Status := RD_LOC_T("DB_Time".ActualTimeDTL);

	    // Convert actual time from DTL format to string
	    "FC_TimeToString"(ia_Date := "DB_Time".ActualTimeDTL,
	                      qs_Date => "DB_Time".ActualTime);

	END_REGION

	REGION 5 – Software version
	    //Function to detect changes in the software and retun software version

	    #sFB_SoftVersion(is_ActualDateTime := "DB_Time".ActualTime,
	                     qs_SoftVersion => "DB_SoftwareVersion".Version,
	                     qa_StandardCRC => "DB_SoftwareVersion".StandardChecksum,
	                     qa_SafetyCRC => "DB_SoftwareVersion".SafetyChecksum);

	END_REGION

	REGION 6 – Profinet diagnostic

	    // CPU Interface 1 HW ID = 262
	    #sFB_ProfiDiag_Net1(iui_LADDR := "DB_Memory"."Local~PROFINET_IO-System",
	                        ix_ExternalScan := FALSE,
	                        qx_ProfinetOk => #sx_ProfiDiag_Net1_OK,
	                        qx_Error => #sx_Error,
	                        iqUDT_EquipmentControl := "DB_Control".System1,
	                        iqUDT_PNDiagArray := "DB_ProfinetDiagnostic".ProfinetNetworks[1],
	                        iqUDT_Statistics := "DB_Statistics".System.Profinet);

	    //Keep only the in use ones.

	    //Network 2 - CM Card 1542-1_1 HW ID = xxxx
	    #sFB_ProfiDiag_Net2(iui_LADDR := #tui_LADDR,
	                        ix_ExternalScan := FALSE,
	                        qx_ProfinetOk => #sx_ProfiDiag_Net2_OK,
	                        qx_Error => #sx_Error,
	                        iqUDT_EquipmentControl := "DB_Control".System1,
	                        iqUDT_PNDiagArray := "DB_ProfinetDiagnostic".ProfinetNetworks[2],
	                        iqUDT_Statistics := "DB_Statistics".System.Profinet);

	    //Network 3 - CM Card 1542-1_2 HW ID = xxxx
	    #sFB_ProfiDiag_Net3(iui_LADDR := #tui_LADDR,
	                        ix_ExternalScan := FALSE,
	                        qx_ProfinetOk => #sx_ProfiDiag_Net3_OK,
	                        qx_Error => #sx_Error,
	                        iqUDT_EquipmentControl := "DB_Control".System1,
	                        iqUDT_PNDiagArray := "DB_ProfinetDiagnostic".ProfinetNetworks[3],
	                        iqUDT_Statistics := "DB_Statistics".System.Profinet);

	    //Network 4 - CM Card 1542-1_3 HW ID = xxxx
	    #sFB_ProfiDiag_Net4(iui_LADDR := #tui_LADDR,
	                        ix_ExternalScan := FALSE,
	                        qx_ProfinetOk => #sx_ProfiDiag_Net4_OK,
	                        qx_Error => #sx_Error,
	                        iqUDT_EquipmentControl := "DB_Control".System1,
	                        iqUDT_PNDiagArray := "DB_ProfinetDiagnostic".ProfinetNetworks[4],
	                        iqUDT_Statistics := "DB_Statistics".System.Profinet);

	    //Network 5 - CM Card 1542-1_4 HW ID = xxxx
	    #sFB_ProfiDiag_Net5(iui_LADDR := #tui_LADDR,
	                        ix_ExternalScan := FALSE,
	                        qx_ProfinetOk => #sx_ProfiDiag_Net5_OK,
	                        qx_Error => #sx_Error,
	                        iqUDT_EquipmentControl := "DB_Control".System1,
	                        iqUDT_PNDiagArray := "DB_ProfinetDiagnostic".ProfinetNetworks[5],
	                        iqUDT_Statistics := "DB_Statistics".System.Profinet);

	    //Network 6 - CM Card 1542-1_5 HW ID = xxxx
	    #sFB_ProfiDiag_Net6(iui_LADDR := #tui_LADDR,
	                        ix_ExternalScan := FALSE,
	                        qx_ProfinetOk => #sx_ProfiDiag_Net6_OK,
	                        qx_Error => #sx_Error,
	                        iqUDT_EquipmentControl := "DB_Control".System1,
	                        iqUDT_PNDiagArray := "DB_ProfinetDiagnostic".ProfinetNetworks[6],
	                        iqUDT_Statistics := "DB_Statistics".System.Profinet);

	    //Network 7 - CM Card 1542-1_6 HW ID = xxxx
	    #sFB_ProfiDiag_Net7(iui_LADDR := #tui_LADDR,
	                        ix_ExternalScan := FALSE,
	                        qx_ProfinetOk => #sx_ProfiDiag_Net7_OK,
	                        qx_Error => #sx_Error,
	                        iqUDT_EquipmentControl := "DB_Control".System1,
	                        iqUDT_PNDiagArray := "DB_ProfinetDiagnostic".ProfinetNetworks[7],
	                        iqUDT_Statistics := "DB_Statistics".System.Profinet);

	    //Network 8 - CM Card 1542-1_7 HW ID = xxxx
	    #sFB_ProfiDiag_Net8(iui_LADDR := #tui_LADDR,
	                        ix_ExternalScan := FALSE,
	                        qx_ProfinetOk => #sx_ProfiDiag_Net8_OK,
	                        qx_Error => #sx_Error,
	                        iqUDT_EquipmentControl := "DB_Control".System1,
	                        iqUDT_PNDiagArray := "DB_ProfinetDiagnostic".ProfinetNetworks[8],
	                        iqUDT_Statistics := "DB_Statistics".System.Profinet);

	    //Network 9 - CM Card 1542-1_8 HW ID = xxxx
	    #sFB_ProfiDiag_Net9(iui_LADDR := #tui_LADDR,
	                        ix_ExternalScan := FALSE,
	                        qx_ProfinetOk => #sx_ProfiDiag_Net9_OK,
	                        qx_Error => #sx_Error,
	                        iqUDT_EquipmentControl := "DB_Control".System1,
	                        iqUDT_PNDiagArray := "DB_ProfinetDiagnostic".ProfinetNetworks[9],
	                        iqUDT_Statistics := "DB_Statistics".System.Profinet);

	    //Network 10 - CM Card 1542-1_9 HW ID = xxxx
	    #sFB_ProfiDiag_Net10(iui_LADDR := #tui_LADDR,
	                         ix_ExternalScan := FALSE,
	                         qx_ProfinetOk => #sx_ProfiDiag_Net10_OK,
	                         qx_Error => #sx_Error,
	                         iqUDT_EquipmentControl := "DB_Control".System1,
	                         iqUDT_PNDiagArray := "DB_ProfinetDiagnostic".ProfinetNetworks[10],
	                         iqUDT_Statistics := "DB_Statistics".System.Profinet);


	END_REGION

	REGION 7 – Profinet OK detection

	    IF #sx_ProfiDiag_Net1_OK
	        AND #sx_ProfiDiag_Net2_OK   //delete if not in use
	        AND #sx_ProfiDiag_Net3_OK   //delete if not in use
	        AND #sx_ProfiDiag_Net4_OK   //delete if not in use
	        AND #sx_ProfiDiag_Net5_OK   //delete if not in use
	        AND #sx_ProfiDiag_Net6_OK   //delete if not in use
	        AND #sx_ProfiDiag_Net7_OK   //delete if not in use
	        AND #sx_ProfiDiag_Net8_OK   //delete if not in use
	        AND #sx_ProfiDiag_Net9_OK   //delete if not in use
	        AND #sx_ProfiDiag_Net10_OK  //delete if not in use
	    THEN

	        "DB_Memory".ScanProfinet := FALSE;

	    END_IF;

	END_REGION
END_FUNCTION_BLOCK

FUNCTION_BLOCK "FB_Communication"
TITLE = FB_Communication
{ S7_Optimized_Access := 'TRUE' }
AUTHOR : MHSE
FAMILY : Communication
VERSION : 3.0
// ATTRIBUTES
// AUTO_NUMBER = True
// BLOCK_NUMBER = 2
// END_ATTRIBUTES
//Function block to handle communication.
   VAR
      sx_Connected { ExternalAccessible := 'False'; ExternalVisible := 'False'; ExternalWritable := 'False'} : Bool;   // TCPIP connection established
   END_VAR


BEGIN
	(*
	----------------------------------------------------------------------------------------
	|                                                                                      |
	|  Copyright  2019             MHS                                                     |
	|  All Rights Reserved         Larenweg 90                                             |
	|                              5234 KC 's-Hertogenbosch,                               |
	|                              Netherlands                                             |
	|                                                                                      |
	----------------------------------------------------------------------------------------

	Version history:
	Date        | Version   | Author        | Remark
	----------------------------------------------------------------------------------------
	24/05/2019  | 0.1       | L.Klar        | first release MHS TIA 15.1
	24/07/2019  | 2.0       | L.Klar        | 2.0 MHS library release TIA 15.1
	23/10/2019  | 2.1       | L.Klar        | FIFO access changed
	23/10/2019  | 2.2       | S.Theocharis  | System number 1 added
	04/11/2019  | 2.3       | L.Klar        | Reconnect command bit changed from memory to DB variable
	12/11/2019  | 3.0       | P.Majka       | 3.0 MHS library release TIA 15.1
	21/02/2023  | 4.0       | F.Baten       | 4.0 Release TIA 17.5
	*)

	REGION Step 1 – Connection initialization

	    "DI_TCPIPConnect"(iUDT_Connection := "DB_Configuration".System.Connection,
	                      qUDT_HMIStatus => "DB_Status".Communication.TCPIPConnect,
	                      qUDT_Status => "DB_CommonStatus".Communication.TCPIPConnect,
	                      iqUDT_EquipmentControl := "DB_Control".System1,
	                      iqUDT_Statistics := "DB_Statistics".Communication.TCPIPConnect,
	                      qx_Connected => #sx_Connected,
	                      iqx_Reconnect := "DB_Memory".ReconnectCommand);

	END_REGION

	REGION Step 2 – Receive data

	    "DI_TCPIPReceive"(iUDT_Connection := "DB_Configuration".System.Connection,
	                      ix_EnableReceive := #sx_Connected,
	                      qx_Error => "DB_ParametrizationErrors".System.Communication.TCPIPReceiveError,
	                      qx_Warning => "DB_ParametrizationErrors".System.Communication.TCPIPReceiveWarning,
	                      iqUDT_FifoHeader := "DB_FIFORcvMsg".Header,
	                      iqa_FifoData := "DB_FIFORcvMsg".Data,
	                      iqUDT_Statistics := "DB_Statistics".Communication.TCPIPReceive);


	END_REGION

	REGION Step 3 – Send data

	    "DI_TCPIPSend"(iUDT_Connection := "DB_Configuration".System.Connection,
	                   ix_EnableSend := #sx_Connected,
	                   qx_Error => "DB_ParametrizationErrors".System.Communication.TCPIPSendError,
	                   qx_Warning => "DB_ParametrizationErrors".System.Communication.TCPIPSendWarning,
	                   iqUDT_FifoLowHeader := "DB_FIFOLowPrioMsg".Header,
	                   iqs_FifoLowData := "DB_FIFOLowPrioMsg".Data,
	                   iqUDT_FifoMedHeader := "DB_FIFOMedPrioMsg".Header,
	                   iqs_FifoMedData := "DB_FIFOMedPrioMsg".Data,
	                   iqUDT_FifoHighHeader := "DB_FIFOHighPrioMsg".Header,
	                   iqs_FifoHighData := "DB_FIFOHighPrioMsg".Data);

	END_REGION
END_FUNCTION_BLOCK

